// TIA Portal project "PID_TANK" (V17)

(* hardware
DEVICE "S71500/ET200MP-Station_1"  S7-1500 station
   slot 0: "Profilschiene_0"  6ES7 590-1***0-0AA0
   slot 1: "PLC_1"  CPU 1511-1 PN  6ES7 511-1AK00-0AB0  V1.8
   slot 2: "AI 8xU/I/RTD/TC ST_1"  AI 8xU/I/RTD/TC ST  6ES7 531-7KF00-0AB0  V2.0
   slot 3: "AI 8xU/I/RTD/TC ST_2"  AI 8xU/I/RTD/TC ST  6ES7 531-7KF00-0AB0  V2.0
   slot 4: "AI 8xU/I/RTD/TC ST_3"  AI 8xU/I/RTD/TC ST  6ES7 531-7KF00-0AB0  V2.0
   slot 5: "AI 8xU/I/RTD/TC ST_4"  AI 8xU/I/RTD/TC ST  6ES7 531-7KF00-0AB0  V2.0
   slot 6: "DI 16x24VDC BA_1"  DI 16x24VDC BA  6ES7 521-1BH10-0AA0  V1.0
   slot 7: "AQ 4xU/I ST_1"  AQ 4xU/I ST  6ES7 532-5HD00-0AB0  V2.2
DEVICE "HMI_1"  TP900 Comfort
   slot 0: "HMI_1"  TP900 Comfort  6AV2 124-0JC01-0AX0  17.0.0.0
   slot 1: "HMI_RT_1"  TP900 Comfort  6AV2 124-0JC01-0AX0  17.0.0.0
   slot 5: "HMI_1.IE_CP_1"  PROFINET Interface  17.0.0.0
      slot 1: "PROFINET Interface_1"  PROFINET Interface
         slot 1: "Port_1"  Port
         slot 2: "Port_2"  Port
   slot 7: "HMI_1.MPI/DP_CP_1"  MPI/DP Interface  17.0.0.0
*)

// ===== PLC "PLC_1"  CPU 1511-1 PN =====

VAR_GLOBAL   // PLC tag table "Standard-Variablentabelle"
   "Tag_1" AT %E0.0 : Bool;
   "Tag_2" AT %Q30.0 : Bool;
   "Tag_3" AT %E0.1 : Bool;
   "Level Meter Sensor" AT %IW30 : Int;
   "Fill Valve Sim" AT %QW30 : Int;
END_VAR

DATA_BLOCK "Tank_DB"   // DB1
{ S7_Optimized_Access := 'TRUE' }
VERSION : 0.1
   VAR
      Setpoint : Int;
      "Level Meter" : Int;
      "Fill Valve" : Int;
      Level_Percentage : Real;
      Liquid_Level : Real;
   END_VAR
BEGIN
END_DATA_BLOCK

FUNCTION "MHJ-PLC-Lab-Function-S71500" : Void   // FC9000, SCL
{ S7_Optimized_Access := 'TRUE' }
VERSION : 0.1
   VAR_TEMP
      Value : Byte;
      ForCounter : Int;
   END_VAR
   VAR CONSTANT
      Value_01_DW : DWord := 16#1223_5486;
      Value_02_DW : DWord := 16#A6C9_D1F5;
   END_VAR
BEGIN

   #Value:=PEEK(area := 16#82,
        dbNumber := 0,
        byteOffset := 511);
   #Value := #Value + 1;

   POKE(area := 16#82,
        dbNumber := 0,
        byteOffset := 511,
        value := #Value);

   POKE(area := 16#82,
        dbNumber := 0,
        byteOffset := 1016,
        value := #Value_01_DW);
   POKE(area := 16#82,
        dbNumber := 0,
        byteOffset := 1020,
        value := #Value_02_DW);

   FOR #ForCounter := 0 TO 63 DO
       #Value:=PEEK(area := 16#1,
            dbNumber := 0,
            byteOffset := #ForCounter);
       POKE(area := 16#81,
            dbNumber := 0,
            byteOffset := #ForCounter,
            value := #Value);
   END_FOR;
   #Value := PEEK(area := 16#1,
                  dbNumber := 0,
                  byteOffset := 512);
   POKE(area := 16#82,
        dbNumber := 0,
        byteOffset := 512,
        value := #Value);
END_FUNCTION

ORGANIZATION_BLOCK "Main"   // OB1, LAD, ProgramCycle
TITLE = "Main Program Sweep (Cycle)"
{ S7_Optimized_Access := 'TRUE' }
VERSION : 0.1
   VAR_INPUT
      Initial_Call : Bool;   // Initial call of this OB
      Remanence : Bool;   // =True, if remanent data are available
   END_VAR
BEGIN

REGION Network 1
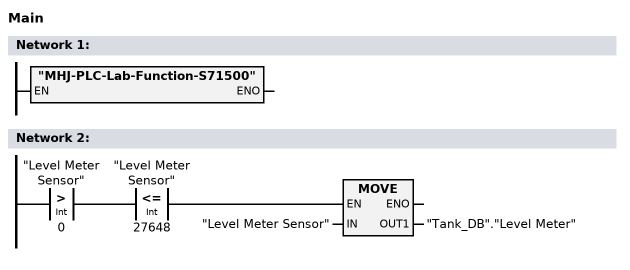
   RUNG wire#powerrail
      "MHJ-PLC-Lab-Function-S71500"()
   END_RUNG
   // the same network as SCL:
   "MHJ-PLC-Lab-Function-S71500"();
END_REGION

REGION Network 2
   RUNG wire#powerrail
      { S7_Templates := "SrcType := Int" } GT_Contact(in1 := "Level Meter Sensor", in2 := 0)
      { S7_Templates := "SrcType := Int" } LE_Contact(in1 := "Level Meter Sensor", in2 := 27648)
      Move(in := "Level Meter Sensor", out1 => "Tank_DB"."Level Meter")
   END_RUNG
   // the same network as SCL:
   IF ("Level Meter Sensor" > 0) AND ("Level Meter Sensor" <= 27648) THEN
       "Tank_DB"."Level Meter" := "Level Meter Sensor";
   END_IF;
END_REGION
END_ORGANIZATION_BLOCK

ORGANIZATION_BLOCK "Cyclic interrupt"   // OB30, LAD, CyclicInterrupt
{ S7_Optimized_Access := 'TRUE' }
VERSION : 0.1
   VAR_INPUT
      Initial_Call : Bool;   // Initial call of this OB
      Event_Count : Int;   // Events discarded
   END_VAR
BEGIN

REGION Network 1
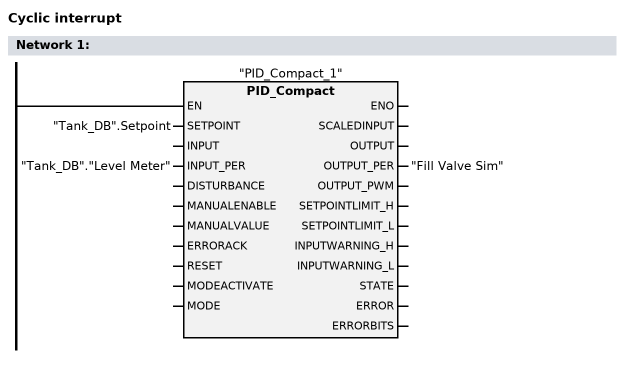
   "PID_Compact_1"(Setpoint := "Tank_DB".Setpoint,   // PID_Compact
                   Input_PER := "Tank_DB"."Level Meter",
                   Output_PER => "Fill Valve Sim");
END_REGION
END_ORGANIZATION_BLOCK

(* ===== HMI "HMI_RT_1" =====
connection "HMI_Connection_1": ETHERNET, S7_1500_OMS

HMI tags "Default tag table"
   "Tank_DB_Setpoint" : Int = PLC Tank_DB.Setpoint, 1 s
   "Tank_DB_Level Meter" : Int = PLC Tank_DB."Level Meter", 1 s
   "Tank_DB_Liquid_Level" : Real = PLC Tank_DB.Liquid_Level, 1 s
   "PID_Compact_1_Retain_CtrlParams_Gain" : Real = PLC PID_Compact_1.Retain.CtrlParams.Gain, 1 s
   "PID_Compact_1_Retain_CtrlParams_Ti" : Real = PLC PID_Compact_1.Retain.CtrlParams.Ti, 1 s
   "PID_Compact_1_Retain_CtrlParams_Td" : Real = PLC PID_Compact_1.Retain.CtrlParams.Td, 1 s

screen "Root screen" 800x480, template "Template_1"
   IOField "I/O field_1" at 378,56 size 60x30; FormatPattern 99
      ProcessValue <- "PID_Compact_1_Retain_CtrlParams_Gain"
   IOField "I/O field_2" at 541,56 size 60x30; FormatPattern 99
      ProcessValue <- "PID_Compact_1_Retain_CtrlParams_Ti"
   IOField "I/O field_3" at 723,56 size 60x30; FormatPattern 99
      ProcessValue <- "PID_Compact_1_Retain_CtrlParams_Td"
   IOField "I/O field_4" at 230,56 size 60x30; FormatPattern 999
      ProcessValue <- "Tank_DB_Setpoint"
   IOField "I/O field_5" at 230,93 size 60x30; FormatPattern 999
      ProcessValue <- "Tank_DB_Level Meter"
   TextField "Text field_1" at 17,56 size 102x27; Text 'Setpoint:'
   TextField "Text field_2" at 17,92 size 226x27; Text 'Current Liquid Level:'
   TextField "Text field_3" at 318,56 size 60x27; Text 'Gain:'
   TextField "Text field_4" at 449,56 size 98x27; Text 'Integral:'
   TextField "Text field_5" at 614,56 size 120x27; Text 'Derivative:'
   TrendView "Trend view_1" at 290,141 size 500x332
   Bar "Bar_1" at 106,138 size 94x338; MinimumValue 0; MaximumValue 300
      ProcessValue <- "Tank_DB_Level Meter"
*)